(* convert value from 64-bit T_FILETIME to 64-bit T_ULARGE_INTEGER *)
FUNCTION F_FILE_FileTimeToULarge : T_ULARGE_INTEGER
VAR_INPUT
	sFileTime		: T_FILETIME;
END_VAR
VAR
END_VAR
(*
-------------------------------------------------------------------------------------------------
Date		Version	Author	Comments
-------------------------------------------------------------------------------------------------
26/03/2012	1.38.00	PB		Initial release

-------------------------------------------------------------------------------------------------
*)

MEMMOVE(ADR(F_FILE_FileTimeToULarge), ADR(sFileTime), SIZEOF(F_FILE_FileTimeToULarge));

END_FUNCTION

(* stored: Version 1.1.0.1, ProductVersion 3.1.4024.15
   POU F_FILE_FileTimeToULarge: Id {eb9ddf76-162b-454f-bce8-d456beb5cbae}, SpecialFunc None *)
